PROGRAM P_StablePlatform
VAR
	fbpA 		: FB_AnalogInputScaling;
	fbpB 		: FB_AnalogInputScaling;
	fbpS 	 	: FB_AnalogInputScaling;
	fSVFeedback : FB_AnalogInputScaling;
	fbPistonPos	: FB_AnalogInputScaling_1;
	fbPistonVel	: FB_AnalogInputScaling_1;
	fbJoystick  : FB_JoystickInputScaling;
	fbSVOutput 	: FB_ValveOutput;
	fbAutoModeControl : FB_AutoModeControl; 
	fbLowPassFilter		: FB_LowpassFilter;
END_VAR

// Enable
IF G_StablePlatformIO.bEnable AND G_StablePlatformIO.bEMG_OK THEN
	G_StablePlatformIO.bActivated := TRUE;
ELSE	
	G_StablePlatformIO.bActivated := FALSE;
END_IF
// Mode
IF G_StablePlatformIO.bActivated AND G_StablePlatformIO.bModeSelector AND  G_Inputs.bAutoModeSelector THEN
	G_StablePlatformIO.bAutoMode := TRUE;
	G_StablePlatformIO.bManualMode := FALSE;
	G_StablePlatformIO.fControlSignal :=  G_StablePlatformIO.fAutoModeControlSignal;
ELSIF G_StablePlatformIO.bActivated AND NOT(G_StablePlatformIO.bModeSelector) AND G_Inputs.bManualModeSelector THEN
	G_StablePlatformIO.bAutoMode := FALSE;
	G_StablePlatformIO.bManualMode := TRUE; 
	G_StablePlatformIO.fControlSignal := -G_StablePlatformScaledIO.fJoystickNormalizedX; 	
ELSE
	G_StablePlatformIO.bAutoMode := FALSE;
	G_StablePlatformIO.bManualMode := FALSE; 
	G_StablePlatformIO.fControlSignal := 0.0;
END_IF

// Inputs
fbpA(
	nRawInput := G_StablePlatformIO.npA,
	stAnalogInputScaling := G_StablePlatformParameters.stPressureSensorScaling400bar,
	fOutput => G_StablePlatformScaledIO.bpA
);

fbpB(
	nRawInput := G_StablePlatformIO.npB,
	stAnalogInputScaling := G_StablePlatformParameters.stPressureSensorScaling400bar,
	fOutput => G_StablePlatformScaledIO.bpB
);

fbpS(
	nRawInput := G_StablePlatformIO.npS,
	stAnalogInputScaling := G_StablePlatformParameters.stPressureSensorScaling400bar,
	fOutput => G_StablePlatformScaledIO.bpS
);

fSVFeedback(
	nRawInput := G_StablePlatformIO.nSVFeedback,
	stAnalogInputScaling := G_StablePlatformParameters.stSVFeedbackScaling,
	fOutput => G_StablePlatformScaledIO.fSVFeedback
);

G_StablePlatformScaledIO.fPlatformAngleDeg := F_rad2deg(G_StablePlatformScaledIO.fPlatformAngle);

// Manual Control

fbJoystick(
	bEnable := G_StablePlatformIO.bManualMode,
	nRawInput := G_Inputs.stJoyLX.nValue,
	stJoystickInputScaling := G_StablePlatformParameters.stJoystickInputScalingX,
	fNormalizedOutput => G_StablePlatformScaledIO.fJoystickNormalizedX
);

// Automode Control
fbAutoModeControl(
	bEnable := G_StablePlatformIO.bAutoMode,
	bModeSelector := G_StablePlatformIO.bMotionModeSelector,
	fSampleTime := G_MachineControl.fSampleTime,
	fPistonPosition := G_StablePlatformScaledIO.fPistionPosFiltered,
	fControlSignal => G_StablePlatformIO.fAutoModeControlSignal
);



// Outputs
fbSVOutput(
	bEnable := NOT(G_Inputs.bRedButton) AND G_StablePlatformIO.bActivated,
	bDeadBandCompOn := FALSE,
	stValveDeadBand := G_StablePlatformParameters.stSVValveDeadBand,
	fNormalizedInput := G_StablePlatformIO.fControlSignal,
	nOutput => G_StablePlatformIO.nSVControlSignal
);

G_StablePlatformIO.bSVEnable := G_StablePlatformIO.bActivated;

fbPistonPos(
	nRawInput := G_StablePlatformIO.nPistonPosition,
	stAnalogInputScaling := G_StablePlatformParameters.stPistonPos,
	fOutput => G_StablePlatformScaledIO.fPistonPosition
);

fbLowPassFilter(
	fInput := G_StablePlatformScaledIO.fPistonPosition,
	fDeltaT := G_MachineControl.fSampleTime,
	fCutoffFreq := G_StablePlatformParameters.fCutoffFreq,
	fDamping := G_StablePlatformParameters.fDamping,
	fOutput => G_StablePlatformScaledIO.fPistionPosFiltered
);

fbPistonVel(
	nRawInput := G_StablePlatformIO.nPistonVelocity,
	stAnalogInputScaling := G_StablePlatformParameters.stPistonVel,
	fOutput => G_StablePlatformScaledIO.fPistonVelocity
);


G_StablePlatformScaledIO.fPlatformAngle := fPlatformAngleTheta1(fStroke:=G_StablePlatformScaledIO.fPistionPosFiltered) + F_deg2rad(G_StablePlatformParameters.fAngleOffsetDeg);

END_PROGRAM

(* stored: Version 1.1.0.1, ProductVersion 3.1.4024.12
   POU P_StablePlatform: Id {c20de7b0-d2cd-4536-8a51-2764cdc32403}, SpecialFunc None *)
